{attribute 'qualified_only'}
VAR_GLOBAL CONSTANT
    cMaxCharacter                   : UDINT(16#FF..16#FFFF) := 16#3FF;          // Default max. character = 1023.
    cMaxProtobufRawBuffer           : UDINT(16#FF..16#FFFF) := 16#1000;         // Default max. raw buffer size = 4096.
    cFieldCodecBytesDefaultSize     : UDINT(16#20..cMaxCharacter) := 16#100;    // Default tmp. buffer size for field codec Bytes.
END_VAR

(* stored: Version 1.1.0.1
   GVL Param_PB: Id {dc2a5d06-2d1d-4ec1-836a-8f032cb5266f}, ParameterList True *)
